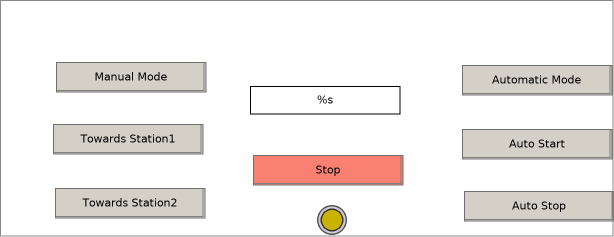
VISUALIZATION Visualization  // 614x237
    Button (56,62 150x30), "Manual Mode"
        tap Control_SFC.iSetManual
    Button (53,124 150x30), "Towards Station1"
        tap Control_SFC.iManualLeft
    Button (55,188 150x30), "Towards Station2"
        tap Control_SFC.iManualRight
    Button (462,65 150x30), "Automatic Mode"
        tap Control_SFC.iSetAuto
    Button (462,129 150x30), "Auto Start"
        tap Control_SFC.iAutoStart
    Button (464,191 150x30), "Auto Stop"
        tap Control_SFC.iAutoStop
    Button (253,155 150x30), "Stop"
        tap Control_SFC.iStop
    Rectangle (250,86 150x28), "%s", text variable: Control_SFC.xMode
    Lamp1 (311,203 42x34), style: Lamp-Lamp1-Yellow
END_VISUALIZATION

(* stored: Version 1.1.0.1, ProductVersion 3.1.4024.12
   Visu Visualization: Id {231c8e07-a297-4bce-8b88-b3bed10b1d32} *)
